FUNCTION_BLOCK INTERNAL FB_ProductEjectedState IMPLEMENTS I_State
VAR_INPUT
END_VAR
VAR_OUTPUT
END_VAR
VAR
	pMachine : I_StateMachine;
	afterProductEjectedNext : I_State;
END_VAR

METHOD CustomerTakesCoin : BOOL
END_METHOD

METHOD CustomerTakesProduct : BOOL
ADSLOGSTR(ADSLOG_MSGTYPE_HINT, 'Customer has taken the product.', '');
pMachine.SetState(afterProductEjectedNext);
END_METHOD

PROPERTY Description : STRING
GET
Description := 'Product Ejected';
END_GET
END_PROPERTY

METHOD InsertCoin : BOOL
END_METHOD

METHOD PressButton : BOOL
END_METHOD

METHOD SetTransitionStates
VAR_INPUT
	Machine : I_StateMachine;
	AfterProductEjectedNext : I_State;
END_VAR
THIS^.afterProductEjectedNext := AfterProductEjectedNext;
THIS^.pMachine := Machine;
END_METHOD

END_FUNCTION_BLOCK

(* stored: Version 1.1.0.1, ProductVersion 3.1.4022.17
   POU FB_ProductEjectedState: Id {826451e0-85d0-40a3-8e88-772e41875071}, SpecialFunc None
   Method CustomerTakesCoin: Id {cfa6fad7-4f8a-4642-ae3e-d6c15280e48f}
   Method CustomerTakesProduct: Id {51573c52-7302-419d-ab99-ca7e195cda82}
   Property Description: Id {01111630-4049-40c8-930a-71a3140c4d6b}
   Get Get: Id {5588fee4-402d-4236-86a6-238402fa0410}
   Method InsertCoin: Id {d9ac4430-7591-4d79-9de2-37f819dcc17e}
   Method PressButton: Id {434d3a03-36cb-41b1-9115-6c78a3e58fab}
   Method SetTransitionStates: Id {5d3d6feb-dcd4-4ac5-b4fd-f2ebd2133e37} *)
